TYPE ALines_t : Array[1..1000] of BYTE; END_TYPE

(* stored: Version 1.1.0.1, ProductVersion 3.1.4024.3
   DUT ALines_t: Id {94f03b62-4f7d-4880-bde0-3115f7203820} *)
